// TIA Portal V20 export
DATA_BLOCK "DB_Alarms_Safety"   // DB150
// stored: AutoNumber false, InstanceOfName FB_Alarms_Safety, InstanceOfType FB
"FB_Alarms_Safety"
   // VAR
   //    sTimerEmergencyPowLaser : IEC_TIMER;
   // END_VAR
BEGIN
END_DATA_BLOCK
